// TIA Portal project "E03_Scheletro" (V18)

(* hardware
DEVICE "S71500/ET200MP station_1"  S7-1500 station
   slot 0: "Telaio di montaggio_0"  Rack  6ES7 590-1***0-0AA0
   slot 1: "PLC_1"  CPU 1516-3 PN/DP  6ES7 516-3AN01-0AB0  V2.5
      slot 3: "Display CPU_1"  6ES7591-1BA00-0AA0
   slot 2: "DI 32x24VDC HF_1"  DI 32x24VDC HF  6ES7 521-1BL00-0AB0  V2.1
   slot 3: "DQ 32x24VDC/0.5A HF_1"  DQ 32x24VDC/0.5A HF  6ES7 522-1BL01-0AB0  V1.0
   slot 4: "AI 8xU/I/RTD/TC ST_1"  AI 8xU/I/RTD/TC ST  6ES7 531-7KF00-0AB0  V2.1
   slot 5: "AQ 4xU/I ST_1"  AQ 4xU/I ST  6ES7 532-5HD00-0AB0  V2.1
*)

// ===== PLC "PLC_1"  CPU 1516-3 PN/DP =====

VAR_GLOBAL   // PLC tag table "Tabella delle variabili standard"
   "led00" AT %Q0.0 : Bool;
   "led01" AT %Q0.1 : Bool;
   "led02" AT %Q0.2 : Bool;
   "led03" AT %Q0.3 : Bool;
   "led04" AT %Q0.4 : Bool;
   "led05" AT %Q0.5 : Bool;
   "led06" AT %Q0.6 : Bool;
   "led07" AT %Q0.7 : Bool;
   "led10" AT %Q1.0 : Bool;
   "led11" AT %Q1.1 : Bool;
   "led12" AT %Q1.2 : Bool;
   "led13" AT %Q1.3 : Bool;
   "led14" AT %Q1.4 : Bool;
   "led15" AT %Q1.5 : Bool;
   "led16" AT %Q1.6 : Bool;
   "led17" AT %Q1.7 : Bool;
   "led20" AT %Q2.0 : Bool;
   "led21" AT %Q2.1 : Bool;
   "led22" AT %Q2.2 : Bool;
   "led23" AT %Q2.3 : Bool;
   "led24" AT %Q2.4 : Bool;
   "led25" AT %Q2.5 : Bool;
   "led26" AT %Q2.6 : Bool;
   "led27" AT %Q2.7 : Bool;
   "led30" AT %Q3.0 : Bool;
   "led31" AT %Q3.1 : Bool;
   "led32" AT %Q3.2 : Bool;
   "led33" AT %Q3.3 : Bool;
   "led34" AT %Q3.4 : Bool;
   "led35" AT %Q3.5 : Bool;
   "led36" AT %Q3.6 : Bool;
   "led37" AT %Q3.7 : Bool;
END_VAR

DATA_BLOCK "DB_Comandi"   // DB1
{ S7_Optimized_Access := 'TRUE' }
VERSION : 0.1
   VAR
      bStop : Bool;
      bAuto : Bool;
      bMan : Bool;
      bReset : Bool;
      bEmergenza : Bool;
   END_VAR
BEGIN
END_DATA_BLOCK

DATA_BLOCK "DB_Stati"   // DB2
{ S7_Optimized_Access := 'TRUE' }
VERSION : 0.1
   VAR
      sAuto : Bool;
      sStop : Bool;
      sMan : Bool;
      sHome : Bool;
      sAttsaStop : Bool;
      sEmergenza : Bool;
      bIni1 : Bool;
      bIni2 : Bool;
      bRip1 : Bool;
      bRip2 : Bool;
   END_VAR
BEGIN
END_DATA_BLOCK

DATA_BLOCK "DB_Tappe"   // DB3
{ S7_Optimized_Access := 'TRUE' }
VERSION : 0.1
   VAR
      tappeGemma : Int;
      tappeM1 : Int;
      tappeM2 : Int;
   END_VAR
BEGIN
END_DATA_BLOCK

DATA_BLOCK "DB_Variabili"   // DB4
{ S7_Optimized_Access := 'TRUE' }
VERSION : 0.1
   VAR
      timerResetPulsantiSTART : Bool;
      timerResetPulsantiDONE : Bool;
      timerResetPulsantiOUTPUT : Time;
      timerResetPulsantiDURATA : Time;
      timerSTART_1 : Bool;
      timerDONE_1 : Bool;
      timerOUTPUT_1 : Time;
      timerDURATA_1 : Time;
      timerSTART_2 : Bool;
      timerDONE_2 : Bool;
      timerOUTPUT_2 : Time;
      timerDURATA_2 : Time;
      timerSTART_3 : Bool;
      timerDONE_3 : Bool;
      timerOUTPUT_3 : Time;
      timerDURATA_3 : Time;
      timerSTART_4 : Bool;
      timerDONE_4 : Bool;
      timerOUTPUT_4 : Time;
      timerDURATA_4 : Time;
      statoLED : Array[0..31] of Bool;
      contatore : Int;
      i : Int;
   END_VAR
BEGIN
END_DATA_BLOCK

// folder: System blocks/Program resources

DATA_BLOCK "timerResetPulstanti"   // DB5
{ S7_Optimized_Access := 'TRUE' }
AUTHOR : Simatic
FAMILY : IEC
NAME : IEC_TMR
VERSION : 1.0
// stored: InstanceOfName IEC_TIMER
"IEC_TIMER"
BEGIN
END_DATA_BLOCK

DATA_BLOCK "timer_1"   // DB6
{ S7_Optimized_Access := 'TRUE' }
AUTHOR : Simatic
FAMILY : IEC
NAME : IEC_TMR
VERSION : 1.0
// stored: InstanceOfName IEC_TIMER
"IEC_TIMER"
BEGIN
END_DATA_BLOCK

DATA_BLOCK "timer_2"   // DB7
{ S7_Optimized_Access := 'TRUE' }
AUTHOR : Simatic
FAMILY : IEC
NAME : IEC_TMR
VERSION : 1.0
// stored: InstanceOfName IEC_TIMER
"IEC_TIMER"
BEGIN
END_DATA_BLOCK

DATA_BLOCK "timer_3"   // DB8
{ S7_Optimized_Access := 'TRUE' }
AUTHOR : Simatic
FAMILY : IEC
NAME : IEC_TMR
VERSION : 1.0
// stored: InstanceOfName IEC_TIMER
"IEC_TIMER"
BEGIN
END_DATA_BLOCK

DATA_BLOCK "timer_4"   // DB9
{ S7_Optimized_Access := 'TRUE' }
AUTHOR : Simatic
FAMILY : IEC
NAME : IEC_TMR
VERSION : 1.0
// stored: InstanceOfName IEC_TIMER
"IEC_TIMER"
BEGIN
END_DATA_BLOCK

// folder: (top level)

FUNCTION "FC_Gemma" : Void   // FC1, SCL
{ S7_Optimized_Access := 'TRUE' }
VERSION : 0.1
BEGIN
   // Gestisce il funzionamento generico del PLC
   // 
   CASE "DB_Tappe".tappeGemma OF
       0: //Stato di riposo 
           "DB_Stati".sStop := TRUE;
           IF "DB_Comandi".bAuto = TRUE THEN
               "DB_Tappe".tappeGemma := 1;
               "DB_Stati".sAttsaStop := FALSE;
               "DB_Stati".sAuto := FALSE;
               "DB_Stati".sHome := TRUE;
               "DB_Stati".sMan := FALSE;
               "DB_Stati".sStop := FALSE;
           ELSE
               IF "DB_Comandi".bMan = TRUE THEN
                   "DB_Tappe".tappeGemma := 4;
                   "DB_Stati".sAttsaStop := FALSE;
                   "DB_Stati".sAuto := FALSE;
                   "DB_Stati".sHome := FALSE;
                   "DB_Stati".sMan := TRUE;
                   "DB_Stati".sStop := FALSE;
               END_IF;
           END_IF
           ;
       1: //Stato di home
           IF "DB_Stati".bIni1 = TRUE AND "DB_Stati".bIni2 = TRUE THEN
               "DB_Tappe".tappeGemma := 2;
               "DB_Stati".sAttsaStop := FALSE;
               "DB_Stati".sAuto := TRUE;
               "DB_Stati".sHome := FALSE;
               "DB_Stati".sMan := FALSE;
               "DB_Stati".sStop := FALSE;
           END_IF;
       2: //Stato di automatico
           IF "DB_Comandi".bStop = TRUE THEN
               "DB_Tappe".tappeGemma := 3;
               "DB_Stati".sAttsaStop := TRUE;
               "DB_Stati".sAuto := FALSE;
               "DB_Stati".sHome := FALSE;
               "DB_Stati".sMan := FALSE;
               "DB_Stati".sStop := FALSE;
               "DB_Stati".sEmergenza := FALSE;
           END_IF;
       3: //Stato di attesa stop
           IF "DB_Stati".bRip1 = TRUE AND "DB_Stati".bRip2 = TRUE THEN
               "DB_Tappe".tappeGemma := 4;
               "DB_Stati".sAttsaStop := FALSE;
               "DB_Stati".sAuto := FALSE;
               "DB_Stati".sHome := FALSE;
               "DB_Stati".sMan := FALSE;
               "DB_Stati".sStop := TRUE;
               "DB_Stati".sEmergenza := FALSE;
           END_IF;
       4: //Stato di manuale
           IF "DB_Comandi".bStop = TRUE THEN
               "DB_Tappe".tappeGemma := 3;
               "DB_Stati".sAttsaStop := TRUE;
               "DB_Stati".sAuto := FALSE;
               "DB_Stati".sHome := FALSE;
               "DB_Stati".sMan := FALSE;
               "DB_Stati".sStop := TRUE;
               "DB_Stati".sEmergenza := FALSE;
           END_IF;
       5: //Stato di emergenza
           IF "DB_Comandi".bEmergenza = TRUE AND "DB_Stati".sEmergenza = TRUE THEN
               "DB_Tappe".tappeGemma := 0;
               "DB_Stati".sAttsaStop := FALSE;
               "DB_Stati".sAuto := FALSE;
               "DB_Stati".sHome := FALSE;
               "DB_Stati".sMan := FALSE;
               "DB_Stati".sStop := TRUE;
               "DB_Stati".sEmergenza := FALSE;
           END_IF;
   END_CASE;

   //Gestione emergenza
   //
   IF "DB_Comandi".bEmergenza = FALSE THEN
       "DB_Tappe".tappeGemma := 5; //Emergenza
       "DB_Stati".sAttsaStop := FALSE;
       "DB_Stati".sAuto := FALSE;
       "DB_Stati".sHome := FALSE;
       "DB_Stati".sMan := FALSE;
       "DB_Stati".sStop := FALSE;
       "DB_Stati".sEmergenza := TRUE;
   END_IF;
END_FUNCTION

FUNCTION "FC_Grafcet" : Void   // FC2, SCL
{ S7_Optimized_Access := 'TRUE' }
VERSION : 0.1
BEGIN
   //Contiene il programma vero e proprio
   //Imposto bini e brip a TRUE
   //Andranno poi gestiti in base alle ondizioni dell'impianto
   //
   "DB_Stati".bIni1 := TRUE;
   "DB_Stati".bIni2 := TRUE;
   "DB_Stati".bRip1 := TRUE;
   "DB_Stati".bRip2 := TRUE;
   //
   //Gestisco il RESET
   //
   IF "DB_Comandi".bReset = TRUE AND
       "DB_Stati".sStop = TRUE THEN
       //Reimposto le condizioni iniziali solo se la macchina è in STOP
       "DB_Tappe".tappeGemma := 0;
       "DB_Tappe".tappeM1 := 0;
       "DB_Tappe".tappeM2 := 0;
       "DB_Variabili".contatore := 0;
       FOR "DB_Variabili".i := 0 TO 31 DO
           "DB_Variabili".statoLED["DB_Variabili".i]:=FALSE;
       END_FOR;
       //per il mio esempio la variabile contatore indica il led di partenza del gioco di luci
       "DB_Variabili".contatore := 24;
   END_IF;

   //
   //Gestisco il grafcet, in questo caso il gioco di luci
   //
   //Gestisco la tappa 0
   //
   IF "DB_Stati".sAuto = TRUE AND
       "DB_Tappe".tappeM1 = 0 THEN
       "DB_Tappe".tappeM1 := 1; //Sono in automatico e la macchina deve iniziare il ciclo di produzione
   END_IF;
   //
   //Gestisco la tappa 1
   //
   //Sono entrato per la prima volta in TAPPA1
   //
   IF "DB_Stati".sAuto = TRUE AND                      //Se sono in automatico
       "DB_Tappe".tappeM1 = 1 AND                      //e tappa 1 
       "DB_Variabili".timerSTART_1 = FALSE THEN        //e il timer_1 non è ancora partito => Faccio partire il timer e accendo i primi due led
       "DB_Variabili".timerSTART_1 := TRUE;
       "DB_Variabili".statoLED[24] := TRUE;
       "DB_Variabili".statoLED[25] := TRUE;
   END_IF;
   // 
   IF "DB_Variabili".timerDONE_1 = TRUE THEN
       //Resetto il timer
       "DB_Variabili".timerDONE_1 := FALSE;
       "DB_Variabili".timerSTART_1 := FALSE;
       //Spegno i led
       "DB_Variabili".statoLED[24] := FALSE;
       "DB_Variabili".statoLED[25] := FALSE;
       //Passo a tappa2
       "DB_Tappe".tappeM1 := 2;
   END_IF;
   //
   //Gestisco la tappa 2
   //
   //Sono entrato per la prima volta in TAPPA2
   //
   IF "DB_Stati".sAuto = TRUE AND                      
       "DB_Tappe".tappeM1 = 2 AND                       
       "DB_Variabili".timerSTART_2 = FALSE THEN
       "DB_Variabili".timerSTART_2 := TRUE;
       "DB_Variabili".statoLED[26] := TRUE;
       "DB_Variabili".statoLED[27] := TRUE;
   END_IF;
   // 
   IF "DB_Variabili".timerDONE_2 = TRUE THEN
       //Resetto il timer
       "DB_Variabili".timerDONE_2 := FALSE;
       "DB_Variabili".timerSTART_2 := FALSE;
       //Spegno i led
       "DB_Variabili".statoLED[26] := FALSE;
       "DB_Variabili".statoLED[27] := FALSE;
       //Passo a tappa3
       "DB_Tappe".tappeM1 := 3;
   END_IF;
   //
   //Gestisco la tappa 3
   //
   IF "DB_Stati".sAuto = TRUE AND
       "DB_Tappe".tappeM1 = 3 AND
       "DB_Variabili".timerSTART_3 = FALSE THEN
       "DB_Variabili".timerSTART_3 := TRUE;
       "DB_Variabili".statoLED[28] := TRUE;
       "DB_Variabili".statoLED[29] := TRUE;
   END_IF;
   // 
   IF "DB_Variabili".timerDONE_3 = TRUE THEN
       //Resetto il timer
       "DB_Variabili".timerDONE_3 := FALSE;
       "DB_Variabili".timerSTART_3 := FALSE;
       //Spegno i led
       "DB_Variabili".statoLED[28] := FALSE;
       "DB_Variabili".statoLED[29] := FALSE;
       //Passo a tappa4
       "DB_Tappe".tappeM1 := 4;
   END_IF;
   //
   //Gestisco la tappa 4
   //
   IF "DB_Stati".sAuto = TRUE AND
       "DB_Tappe".tappeM1 = 4 AND
       "DB_Variabili".timerSTART_4 = FALSE THEN
       "DB_Variabili".timerSTART_4 := TRUE;
       "DB_Variabili".statoLED[30] := TRUE;
       "DB_Variabili".statoLED[31] := TRUE;
   END_IF;
   // 
   IF "DB_Variabili".timerDONE_4 = TRUE THEN
       //Resetto il timer
       "DB_Variabili".timerDONE_4 := FALSE;
       "DB_Variabili".timerSTART_4 := FALSE;
       //Spegno i led
       "DB_Variabili".statoLED[30] := FALSE;
       "DB_Variabili".statoLED[31] := FALSE;
       //Passo a tappa 1
       "DB_Tappe".tappeM1 := 1;
   END_IF;
END_FUNCTION

FUNCTION "FC_ResetPulsanti" : Void   // FC3, SCL
{ S7_Optimized_Access := 'TRUE' }
VERSION : 0.1
BEGIN
   IF "DB_Comandi".bAuto = TRUE OR
       "DB_Comandi".bMan = TRUE OR
       "DB_Comandi".bReset = TRUE OR
       "DB_Comandi".bStop = TRUE
   THEN
       "DB_Variabili".timerResetPulsantiSTART := TRUE;
   END_IF;

   IF "DB_Variabili".timerResetPulsantiDONE = TRUE THEN
       "DB_Variabili".timerResetPulsantiSTART := FALSE;
       "DB_Variabili".timerResetPulsantiDONE := FALSE;
       "DB_Comandi".bAuto := FALSE;
       "DB_Comandi".bMan := FALSE;
       "DB_Comandi".bReset := FALSE;
       "DB_Comandi".bStop := FALSE;
   END_IF;
END_FUNCTION

FUNCTION "FC_Timer" : Void   // FC4, SCL
{ S7_Optimized_Access := 'TRUE' }
VERSION : 0.1
BEGIN
   "DB_Variabili".timerResetPulsantiDURATA := T#500ms;
   "timerResetPulstanti".TON(IN:="DB_Variabili".timerResetPulsantiSTART,
                             PT:="DB_Variabili".timerResetPulsantiDURATA,
                             Q=>"DB_Variabili".timerResetPulsantiDONE,
                             ET => "DB_Variabili".timerResetPulsantiOUTPUT );
   //
   "DB_Variabili".timerDURATA_1 := T#1000ms;
   "timer_1".TON(IN:="DB_Variabili".timerSTART_1,
                 PT:="DB_Variabili".timerDURATA_1,
                 Q=>"DB_Variabili".timerDONE_1,
                 ET=>"DB_Variabili".timerOUTPUT_1);
   //
   "DB_Variabili".timerDURATA_2 := T#500ms;
   "timer_2".TON(IN:="DB_Variabili".timerSTART_2,
                 PT:="DB_Variabili".timerDURATA_2,
                 Q=>"DB_Variabili".timerDONE_2,
                 ET=>"DB_Variabili".timerOUTPUT_2);
   //
   "DB_Variabili".timerDURATA_3 := T#1500ms;
   "timer_3".TON(IN := "DB_Variabili".timerSTART_3,
                 PT := "DB_Variabili".timerDURATA_3,
                 Q => "DB_Variabili".timerDONE_3,
                 ET => "DB_Variabili".timerOUTPUT_3);
   //
   "DB_Variabili".timerDURATA_4 := T#200ms;
   "timer_4".TON(IN:="DB_Variabili".timerSTART_4,
                 PT:="DB_Variabili".timerDURATA_4,
                 Q=>"DB_Variabili".timerDONE_4,
                 ET=>"DB_Variabili".timerOUTPUT_4);
END_FUNCTION

FUNCTION "FC_Uscite" : Void   // FC5, SCL
{ S7_Optimized_Access := 'TRUE' }
VERSION : 0.1
BEGIN
   //Prima di scrivere fisicamente le uscite devo controllare che tutte le condizioni siano rispettate
   //Emergenza,Protezioni, Fotocellule et cetera..
   //
   "led30" := "DB_Variabili".statoLED[24];
   "led31" := "DB_Variabili".statoLED[25];
   "led32" := "DB_Variabili".statoLED[26];
   "led33" := "DB_Variabili".statoLED[27];
   "led34" := "DB_Variabili".statoLED[28];
   "led35" := "DB_Variabili".statoLED[29];
   "led36" := "DB_Variabili".statoLED[30];
   "led37" := "DB_Variabili".statoLED[31];
END_FUNCTION

ORGANIZATION_BLOCK "Main"   // OB1, LAD, ProgramCycle
TITLE = "Main Program Sweep (Cycle)"
{ S7_Optimized_Access := 'TRUE' }
VERSION : 0.1
   VAR_INPUT
      Initial_Call : Bool;   // Initial call of this OB
      Remanence : Bool;   // =True, if remanent data are available
   END_VAR
   VAR_TEMP   // added for the SCL form of the ladder/FBD networks
      _w1 : Bool;
      _w2 : Bool;
      _w3 : Bool;
      _w4 : Bool;
   END_VAR
BEGIN

REGION Network 1
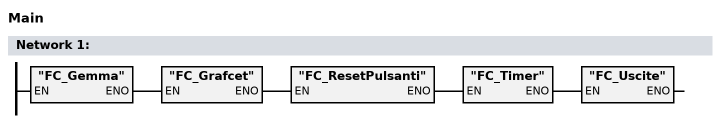
   RUNG wire#powerrail
      "FC_Gemma"()
      "FC_Grafcet"()
      "FC_ResetPulsanti"()
      "FC_Timer"()
      "FC_Uscite"()
   END_RUNG
   // the same network as SCL:
   "FC_Gemma"(ENO => #_w1);
   "FC_Grafcet"(EN := #_w1, ENO => #_w2);
   "FC_ResetPulsanti"(EN := #_w2, ENO => #_w3);
   "FC_Timer"(EN := #_w3, ENO => #_w4);
   IF #_w4 THEN "FC_Uscite"(); END_IF;
END_REGION
END_ORGANIZATION_BLOCK